{attribute addProperty BoxType "EP2328-1061-0016"}
{attribute addProperty Id "OutputAT %Q*BOOL81"}
{attribute addProperty CRC "2134331056"}
{attribute addProperty SizeInBites "8"}
{attribute addProperty SizeInBytes "1"}
TYPE DO_X04_Pin4_Output_7F374EB0 :
STRUCT
	{attribute addProperty Name "Output"}
	Output AT %Q* : BOOL;
END_STRUCT
END_TYPE

(* stored: Version 1.2.0.0, ProductVersion 3.1.4024.9
   DUT DO_X04_Pin4_Output_7F374EB0: Id {0827b3b9-8180-472e-9ac4-645599b35afd} *)
